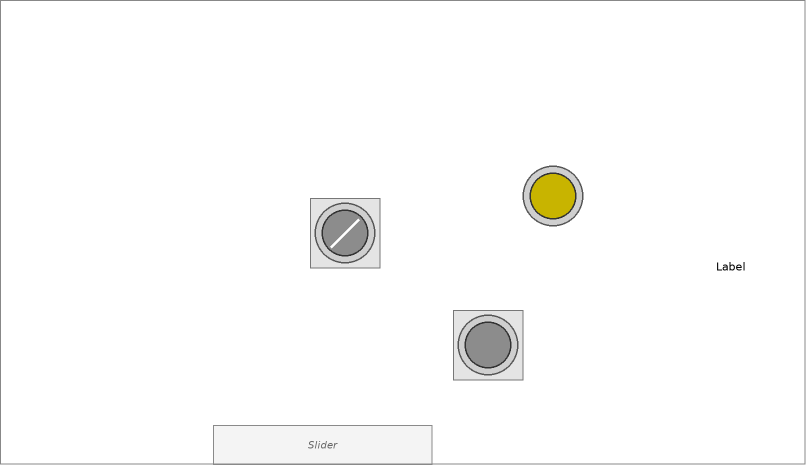
VISUALIZATION HMI  // 806x465
    Lamp1 (518,161 70x70), style: Lamp-Lamp1-Yellow
    RotarySwitch (310,198 70x70), behaviour: TOGGLE, style: Switch-RotarySwitch-Gray
    PushSwitch (453,310 70x70), behaviour: TOGGLE, style: Switch-PushSwitch-Gray
    Label (656,252 150x30), "Label"
    Slider (213,425 219x40), scale 0..100
END_VISUALIZATION

(* stored: Version 1.1.0.1
   Visu HMI: Id {bd73dd53-f30c-4012-bc0c-b203036691d2} *)
